// TIA Portal V19 export
TYPE "LubrValve_ITF"
// stored: Access Published
   STRUCT
      Sts : Struct
         PumpType : Int;   // 0:MotorPump, 1:AirPump
         Running : Bool;
         Error : Bool;
      END_STRUCT;
      Ctrl : Struct
         RstAlarms : Bool;
         WorkReq : Bool;
      END_STRUCT;
      ValveChain : Struct
         ActualValve : Int;
         MaxValve : Int;
      END_STRUCT;
   END_STRUCT;
END_TYPE
